% RSLogix 500 project SENSORCALIBRATION_BAK008.RSS, saved by version 8.30.00.16 %
PROJECT "UNTITLED"    % processor: Bul.1763 MicroLogix 1100 Series B %

PROGRAM FILES
  LAD 2   3 rungs
  LAD 3 "I/O"  4 rungs  % Inputs & Outputs %
  LAD 4 "CONTROLS"  17 rungs  % Control Logic %

DATA FILES
  O0 OUTPUT  4 elements
  I1 INPUT  6 elements
  S2 STATUS  66 elements
  B3 BINARY  2 elements
  T4 TIMER  2 elements
  C5 COUNTER  1 elements
  R6 CONTROL  1 elements
  N7 INTEGER  15 elements
  F8 FLOAT  1 elements
  L9 LONG  5 elements

LADDER 2
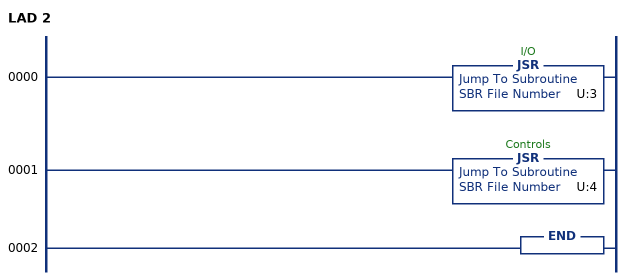
% Rung: 0 %
SOR JSR U:3 EOR
%   U:3  "I/O" %
% Rung: 1 %
SOR JSR U:4 EOR
%   U:4  "Controls" %
% Rung: 2 %
SOR END EOR

LADDER 3 "I/O"    % Inputs & Outputs %
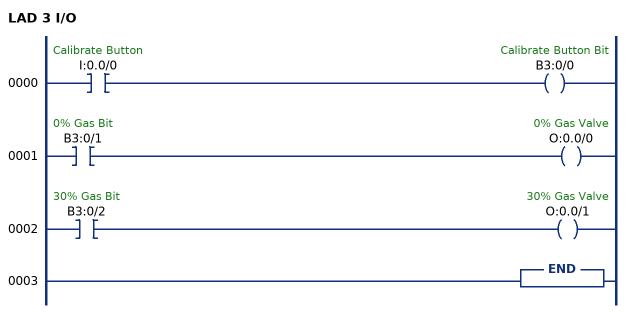
% Rung: 0 %
SOR XIC I:0.0/0 OTE B3:0/0 EOR
%   I:0.0/0  "Calibrate Button" %
%   B3:0/0  "Calibrate Button Bit" %
% Rung: 1 %
SOR XIC B3:0/1 OTE O:0.0/0 EOR
%   B3:0/1  "0% Gas Bit" %
%   O:0.0/0  "0% Gas Valve" %
% Rung: 2 %
SOR XIC B3:0/2 OTE O:0.0/1 EOR
%   B3:0/2  "30% Gas Bit" %
%   O:0.0/1  "30% Gas Valve" %
% Rung: 3 %
SOR END EOR

LADDER 4 "CONTROLS"    % Control Logic %
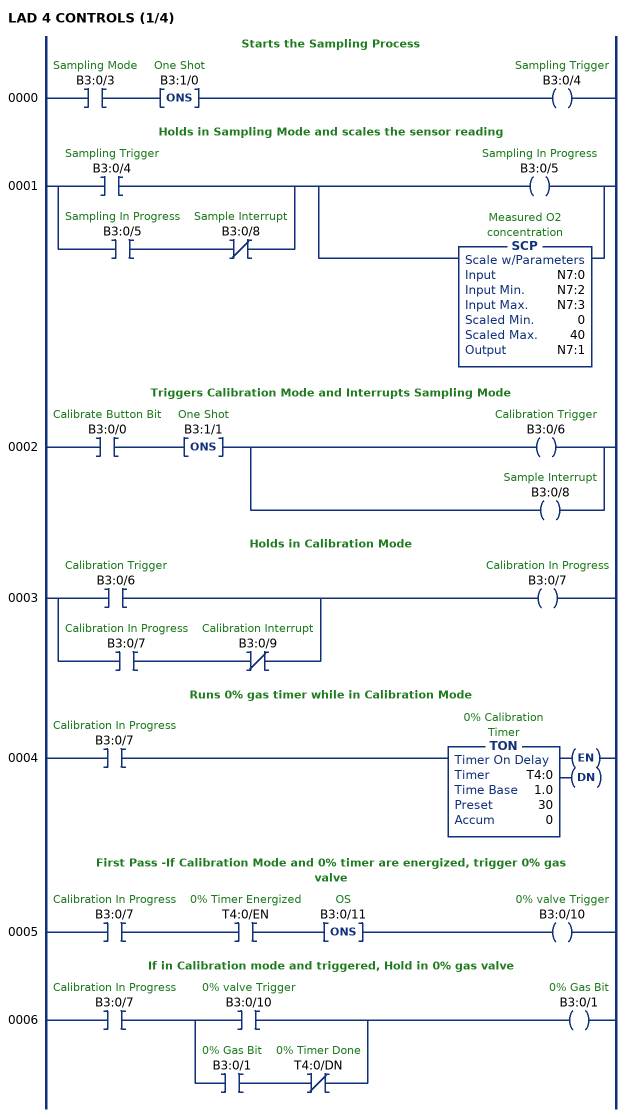
% Rung: 0 %
% TITLE: Starts the Sampling Process %
SOR XIC B3:0/3 ONS B3:1/0 OTE B3:0/4 EOR
%   B3:0/3  "Sampling Mode" %
%   B3:1/0  "One Shot" %
%   B3:0/4  "Sampling Trigger" %
% Rung: 1 %
% TITLE: Holds in Sampling Mode and scales the sensor reading %
SOR BST XIC B3:0/4 NXB XIC B3:0/5 XIO B3:0/8 BND BST OTE B3:0/5 NXB SCP N7:0 N7:2 N7:3 0 40 N7:1 BND EOR
%   B3:0/4  "Sampling Trigger" %
%   B3:0/5  "Sampling In Progress" %
%   B3:0/8  "Sample Interrupt" %
%   N7:0  "O2 Sensor" %
%   N7:2  "Calibrated O2 min" %
%   N7:3  "Calibrated O2 max" %
%   N7:1  "Measured O2 concentration" %
% Rung: 2 %
% TITLE: Triggers Calibration Mode and Interrupts Sampling Mode %
SOR XIC B3:0/0 ONS B3:1/1 BST OTE B3:0/6 NXB OTE B3:0/8 BND EOR
%   B3:0/0  "Calibrate Button Bit" %
%   B3:1/1  "One Shot" %
%   B3:0/6  "Calibration Trigger" %
%   B3:0/8  "Sample Interrupt" %
% Rung: 3 %
% TITLE: Holds in Calibration Mode %
SOR BST XIC B3:0/6 NXB XIC B3:0/7 XIO B3:0/9 BND OTE B3:0/7 EOR
%   B3:0/6  "Calibration Trigger" %
%   B3:0/7  "Calibration In Progress" %
%   B3:0/9  "Calibration Interrupt" %
% Rung: 4 %
% TITLE: Runs 0% gas timer while in Calibration Mode %
SOR XIC B3:0/7 TON T4:0 1.0 30 0 EOR
%   B3:0/7  "Calibration In Progress" %
%   T4:0  "0% Calibration Timer" %
% Rung: 5 %
% TITLE: First Pass -If Calibration Mode and 0% timer are energized, trigger 0% gas valve %
SOR XIC B3:0/7 XIC T4:0/EN ONS B3:0/11 OTE B3:0/10 EOR
%   B3:0/7  "Calibration In Progress" %
%   T4:0/EN  "0% Timer Energized" %
%   B3:0/11  "OS" %
%   B3:0/10  "0% valve Trigger" %
% Rung: 6 %
% TITLE: If in Calibration mode and triggered, Hold in 0% gas valve %
SOR XIC B3:0/7 BST XIC B3:0/10 NXB XIC B3:0/1 XIO T4:0/DN BND OTE B3:0/1 EOR
%   B3:0/7  "Calibration In Progress" %
%   B3:0/10  "0% valve Trigger" %
%   B3:0/1  "0% Gas Bit" %
%   T4:0/DN  "0% Timer Done" %

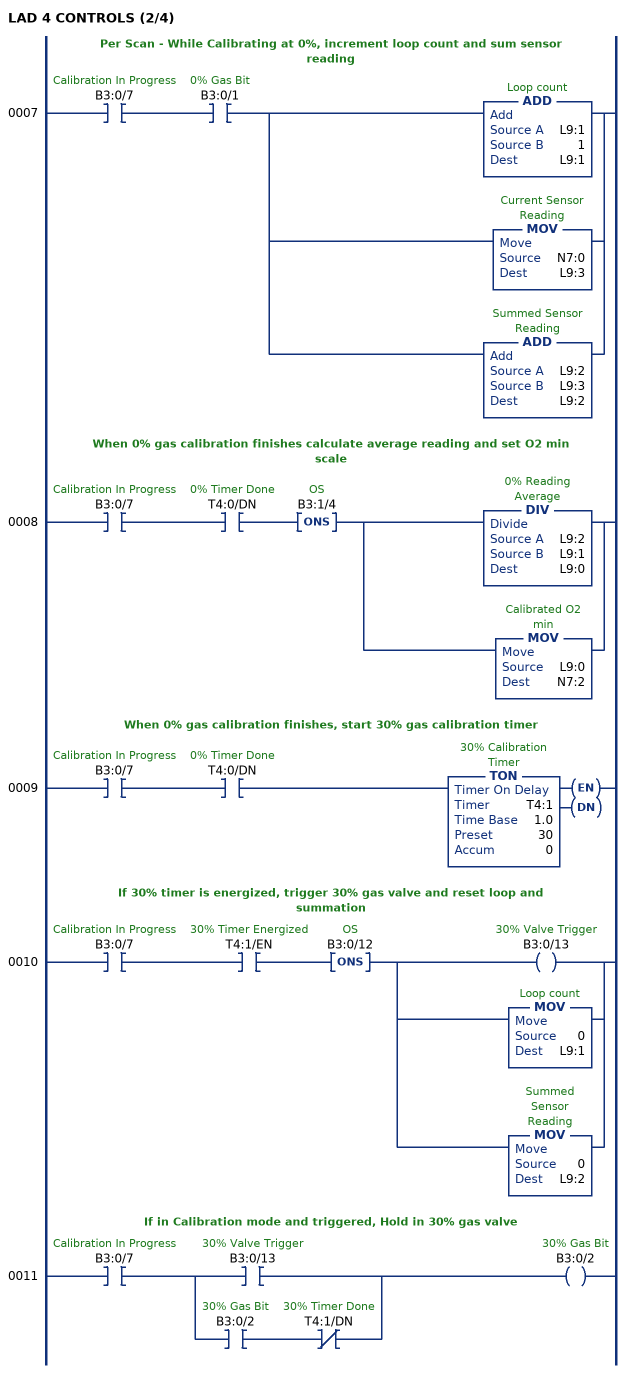
% Rung: 7 %
% TITLE: Per Scan - While Calibrating at 0%, increment loop count and sum sensor reading %
SOR XIC B3:0/7 XIC B3:0/1 BST ADD L9:1 1 L9:1 NXB BST MOV N7:0 L9:3 NXB ADD L9:2 L9:3 L9:2 BND BND EOR
%   B3:0/7  "Calibration In Progress" %
%   B3:0/1  "0% Gas Bit" %
%   L9:1  "Loop count" %
%   N7:0  "O2 Sensor" %
%   L9:3  "Current Sensor Reading" %
%   L9:2  "Summed Sensor Reading" %
% Rung: 8 %
% TITLE: When 0% gas calibration finishes calculate average reading and set O2 min scale %
SOR XIC B3:0/7 XIC T4:0/DN ONS B3:1/4 BST DIV L9:2 L9:1 L9:0 NXB MOV L9:0 N7:2 BND EOR
%   B3:0/7  "Calibration In Progress" %
%   T4:0/DN  "0% Timer Done" %
%   B3:1/4  "OS" %
%   L9:2  "Summed Sensor Reading" %
%   L9:1  "Loop count" %
%   L9:0  "0% Reading Average" %
%   N7:2  "Calibrated O2 min" %
% Rung: 9 %
% TITLE: When 0% gas calibration finishes, start 30% gas calibration timer %
SOR XIC B3:0/7 XIC T4:0/DN TON T4:1 1.0 30 0 EOR
%   B3:0/7  "Calibration In Progress" %
%   T4:0/DN  "0% Timer Done" %
%   T4:1  "30% Calibration Timer" %
% Rung: 10 %
% TITLE: If 30% timer is energized, trigger 30% gas valve and reset loop and summation %
SOR XIC B3:0/7 XIC T4:1/EN ONS B3:0/12 BST OTE B3:0/13 NXB BST MOV 0 L9:1 NXB MOV 0 L9:2 BND BND EOR
%   B3:0/7  "Calibration In Progress" %
%   T4:1/EN  "30% Timer Energized" %
%   B3:0/12  "OS" %
%   B3:0/13  "30% Valve Trigger" %
%   L9:1  "Loop count" %
%   L9:2  "Summed Sensor Reading" %
% Rung: 11 %
% TITLE: If in Calibration mode and triggered, Hold in 30% gas valve %
SOR XIC B3:0/7 BST XIC B3:0/13 NXB XIC B3:0/2 XIO T4:1/DN BND OTE B3:0/2 EOR
%   B3:0/7  "Calibration In Progress" %
%   B3:0/13  "30% Valve Trigger" %
%   B3:0/2  "30% Gas Bit" %
%   T4:1/DN  "30% Timer Done" %

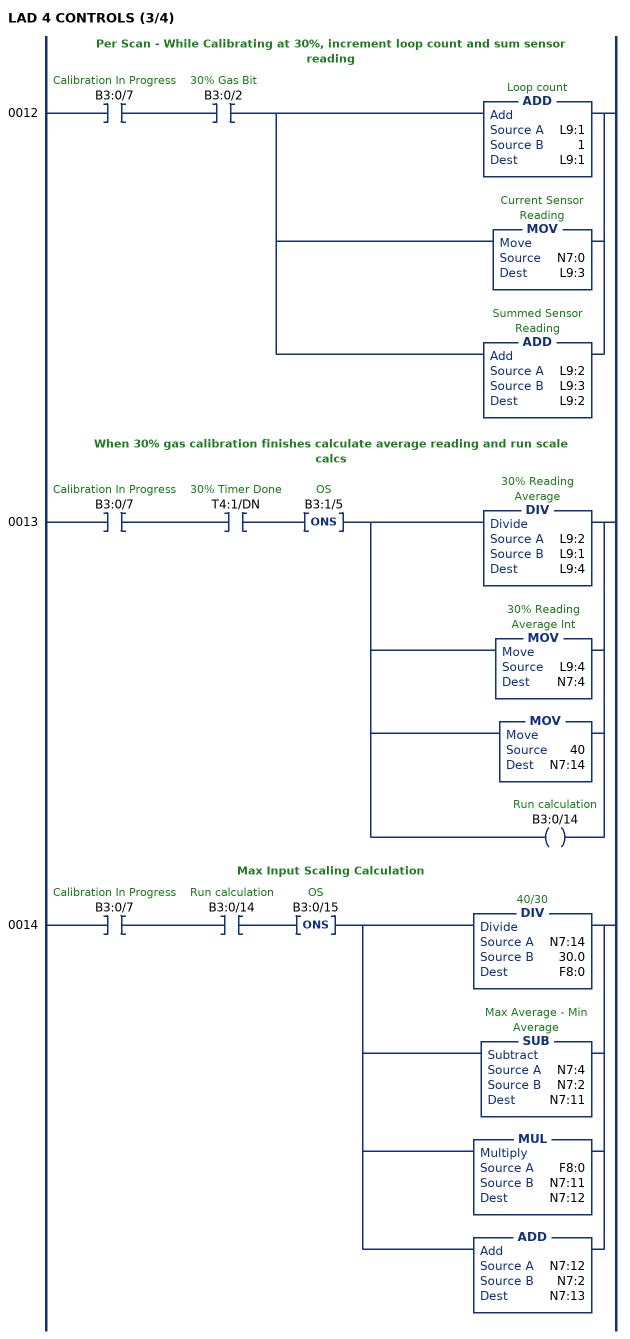
% Rung: 12 %
% TITLE: Per Scan - While Calibrating at 30%, increment loop count and sum sensor reading %
SOR XIC B3:0/7 XIC B3:0/2 BST ADD L9:1 1 L9:1 NXB BST MOV N7:0 L9:3 NXB ADD L9:2 L9:3 L9:2 BND BND EOR
%   B3:0/7  "Calibration In Progress" %
%   B3:0/2  "30% Gas Bit" %
%   L9:1  "Loop count" %
%   N7:0  "O2 Sensor" %
%   L9:3  "Current Sensor Reading" %
%   L9:2  "Summed Sensor Reading" %
% Rung: 13 %
% TITLE: When 30% gas calibration finishes calculate average reading and run scale calcs %
SOR XIC B3:0/7 XIC T4:1/DN ONS B3:1/5 BST DIV L9:2 L9:1 L9:4 NXB BST MOV L9:4 N7:4 NXB BST MOV 40 N7:14 NXB OTE B3:0/14 BND BND BND EOR
%   B3:0/7  "Calibration In Progress" %
%   T4:1/DN  "30% Timer Done" %
%   B3:1/5  "OS" %
%   L9:2  "Summed Sensor Reading" %
%   L9:1  "Loop count" %
%   L9:4  "30% Reading Average" %
%   N7:4  "30% Reading Average Int" %
%   B3:0/14  "Run calculation" %
% Rung: 14 %
% TITLE: Max Input Scaling Calculation %
SOR XIC B3:0/7 XIC B3:0/14 ONS B3:0/15 BST DIV N7:14 30.0 F8:0 NXB BST SUB N7:4 N7:2 N7:11 NXB BST MUL F8:0 N7:11 N7:12 NXB ADD N7:12 N7:2 N7:13 BND BND BND EOR
%   B3:0/7  "Calibration In Progress" %
%   B3:0/14  "Run calculation" %
%   B3:0/15  "OS" %
%   F8:0  "40/30" %
%   N7:4  "30% Reading Average Int" %
%   N7:2  "Calibrated O2 min" %
%   N7:11  "Max Average - Min Average" %

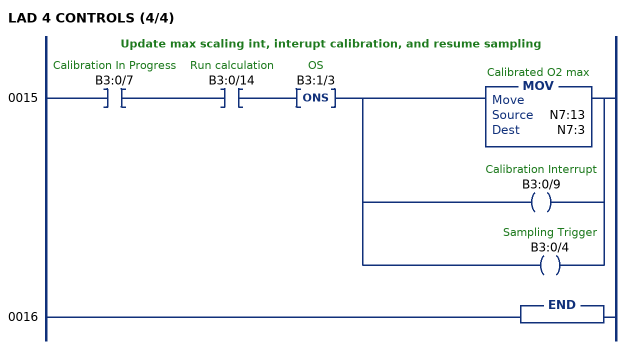
% Rung: 15 %
% TITLE: Update max scaling int, interupt calibration, and resume sampling %
SOR XIC B3:0/7 XIC B3:0/14 ONS B3:1/3 BST MOV N7:13 N7:3 NXB BST OTE B3:0/9 NXB OTE B3:0/4 BND BND EOR
%   B3:0/7  "Calibration In Progress" %
%   B3:0/14  "Run calculation" %
%   B3:1/3  "OS" %
%   N7:3  "Calibrated O2 max" %
%   B3:0/9  "Calibration Interrupt" %
%   B3:0/4  "Sampling Trigger" %
% Rung: 16 %
SOR END EOR

OTHER DOCUMENTED ADDRESSES
  B3:1/2  "One Shot"
  L9:5  "Summed Sensor reading"
  N7:5  "Did run?"
  N7:6  "0& calibration value"
  N7:7  "30% loop count"
  N7:9  "30% calibration value"

COMMENTS NOT ATTACHED TO A CURRENT RUNG
  B3:0/1: If in Calibration mode and triggered, Hold in 0% gas valve
  B3:0/10: First Pass -If Calibration Mode and 0% timer are energized, trigger 0% gas valve
  T4:0: Runs 0% gas timer while in Calibration Mode
  B3:0/7: Holds in Calibration Mode
  B3:0/8: Triggers Calibration Mode and Interrupts Sampling Mode
  N7:1: Holds in Sampling Mode and scales the sensor reading
  B3:0/2: If in Calibration mode and triggered, Hold in 30% gas valve
  T4:1: When 0% gas calibration finishes, start 30% gas calibration timer
  N7:2: When 0% gas calibration finishes calculate average reading and set O2 min scale

DATA TABLE (non-zero values as saved)
DATA T4
% .PRE .ACC %
% T4:0 % 30 0
% T4:1 % 30 0
